(* CoDeSys 2.3 project: forGomon.pro *)
(* Libraries: esx_ioxp.lib*19.12.13 12:14:40, Standard.lib 4.10.05 11:14:46 *)

(* PLC configuration (modules and I/O channels)
gq_Ignition AT %IX0.0 [X_SYS_IGNITION] Ignition pin (D+)
gs16_TempBoard AT %IW1 [X_SYS_TEMP_BOARD] System temperature in degree Celsius
gu32_TimeMs AT %ID1 [X_SYS_TIME_MS] System time in ms
gq_StayAlive AT %QX0.0 [X_SYS_STAY_ALIVE] Stay alive mechanism
gq_Relay AT %QX1.0 [X_SYS_RELAY_1] Safety relay
gs32_SensorSupply AT %QD1 [X_SYS_SENSOR_SUPPLY_1] External sensor supply
gs32_IO01 AT %QD2 [InOut] IO01, PIN 9 (PWM H/L, DO, CC, VIN (40V), DIN) {InOut_Type = uninitialized; InOut_FilterConfig = 0; InOut_Circuit1 = X_IN_CIRCUIT_ACTIVE_HIGH; InOut_Circuit2 = X_IN_CIRCUIT_NO_PULL_UP; PWM_MaxValue = 10000}
gs32_IO02 AT %QD3 [InOut] IO02, PIN 8 (PWM H/L, DO, CC, VIN (40V), DIN) {InOut_Type = uninitialized; InOut_FilterConfig = 0; InOut_Circuit1 = X_IN_CIRCUIT_ACTIVE_HIGH; InOut_Circuit2 = X_IN_CIRCUIT_NO_PULL_UP; PWM_MaxValue = 10000}
gs32_IO03 AT %QD4 [InOut] IO03, PIN 7 (PWM H/L, DO, CC, VIN (40V), DIN) {InOut_Type = uninitialized; InOut_FilterConfig = 0; InOut_Circuit1 = X_IN_CIRCUIT_ACTIVE_HIGH; InOut_Circuit2 = X_IN_CIRCUIT_NO_PULL_UP; PWM_MaxValue = 10000}
gs32_IO04 AT %QD5 [InOut] IO04, PIN 6 (PWM H/L, DO, CC, VIN (40V), DIN) {InOut_Type = uninitialized; InOut_FilterConfig = 0; InOut_Circuit1 = X_IN_CIRCUIT_ACTIVE_HIGH; InOut_Circuit2 = X_IN_CIRCUIT_NO_PULL_UP; PWM_MaxValue = 10000}
gs32_IO05 AT %QD6 [InOut] IO05, PIN 13 (PWM H, DO, DIN) {InOut_Type = uninitialized; InOut_FilterConfig = 0; InOut_Circuit1 = X_IN_CIRCUIT_ACTIVE_HIGH; InOut_Circuit2 = X_IN_CIRCUIT_NO_PULL_UP; PWM_MaxValue = 10000}
gs32_IO06 AT %QD7 [InOut] IO06, PIN 12 (PWM H, DO, DIN) {InOut_Type = uninitialized; InOut_FilterConfig = 0; InOut_Circuit1 = X_IN_CIRCUIT_ACTIVE_HIGH; InOut_Circuit2 = X_IN_CIRCUIT_NO_PULL_UP; PWM_MaxValue = 10000}
gs32_IO07 AT %QD8 [InOut] IO07, PIN 11 (PWM H, DO, DIN) {InOut_Type = uninitialized; InOut_FilterConfig = 0; InOut_Circuit1 = X_IN_CIRCUIT_ACTIVE_HIGH; InOut_Circuit2 = X_IN_CIRCUIT_NO_PULL_UP; PWM_MaxValue = 10000}
gs32_IO08 AT %QD9 [InOut] IO08, PIN 10 (PWM H, DO, DIN) {InOut_Type = uninitialized; InOut_FilterConfig = 0; InOut_Circuit1 = X_IN_CIRCUIT_ACTIVE_HIGH; InOut_Circuit2 = X_IN_CIRCUIT_NO_PULL_UP; PWM_MaxValue = 10000}
gs32_IO09 AT %ID2 [InOut] IO09, PIN 2 (DIN, FIN, IIN) {InOut_Type = uninitialized; InOut_FilterConfig = 0; InOut_Circuit1 = X_IN_CIRCUIT_ACTIVE_HIGH; InOut_Circuit2 = X_IN_CIRCUIT_NO_PULL_UP; PWM_MaxValue = 10000}
gs32_IO10 AT %ID3 [InOut] IO10, PIN 3 (DIN, FIN, IIN) {InOut_Type = uninitialized; InOut_FilterConfig = 0; InOut_Circuit1 = X_IN_CIRCUIT_ACTIVE_HIGH; InOut_Circuit2 = X_IN_CIRCUIT_NO_PULL_UP; PWM_MaxValue = 10000}
gs32_IO11 AT %ID4 [InOut] IO11, PIN 4 (DIN, FIN, IIN) {InOut_Type = uninitialized; InOut_FilterConfig = 0; InOut_Circuit1 = X_IN_CIRCUIT_ACTIVE_HIGH; InOut_Circuit2 = X_IN_CIRCUIT_NO_PULL_UP; PWM_MaxValue = 10000}
gs32_IO12 AT %ID5 [InOut] IO12, PIN 5 (DIN) {InOut_Type = uninitialized; InOut_FilterConfig = 0; InOut_Circuit1 = X_IN_CIRCUIT_ACTIVE_HIGH; InOut_Circuit2 = X_IN_CIRCUIT_NO_PULL_UP; PWM_MaxValue = 10000}
gs32_IO13 AT %ID6 [InOut] IO13, PIN 38 (CIN (20mA), DIN) {InOut_Type = uninitialized; InOut_FilterConfig = 0; InOut_Circuit1 = X_IN_CIRCUIT_ACTIVE_HIGH; InOut_Circuit2 = X_IN_CIRCUIT_NO_PULL_UP; PWM_MaxValue = 10000}
gs32_IO14 AT %ID7 [InOut] IO14, PIN 24 (CIN (20mA), DIN) {InOut_Type = uninitialized; InOut_FilterConfig = 0; InOut_Circuit1 = X_IN_CIRCUIT_ACTIVE_HIGH; InOut_Circuit2 = X_IN_CIRCUIT_NO_PULL_UP; PWM_MaxValue = 10000}
gs32_IO15 AT %ID8 [InOut] IO15, PIN 39 (CIN (20mA), DIN) {InOut_Type = uninitialized; InOut_FilterConfig = 0; InOut_Circuit1 = X_IN_CIRCUIT_ACTIVE_HIGH; InOut_Circuit2 = X_IN_CIRCUIT_NO_PULL_UP; PWM_MaxValue = 10000}
gs32_IO16 AT %ID9 [InOut] IO16, PIN 25 (CIN (20mA), DIN) {InOut_Type = uninitialized; InOut_FilterConfig = 0; InOut_Circuit1 = X_IN_CIRCUIT_ACTIVE_HIGH; InOut_Circuit2 = X_IN_CIRCUIT_NO_PULL_UP; PWM_MaxValue = 10000}
gs32_IO17 AT %ID10 [InOut] IO17, PIN 40 (CIN (20mA), DIN) {InOut_Type = uninitialized; InOut_FilterConfig = 0; InOut_Circuit1 = X_IN_CIRCUIT_ACTIVE_HIGH; InOut_Circuit2 = X_IN_CIRCUIT_NO_PULL_UP; PWM_MaxValue = 10000}
gs32_IO18 AT %ID11 [InOut] IO18, PIN 26 (CIN (20mA), DIN) {InOut_Type = uninitialized; InOut_FilterConfig = 0; InOut_Circuit1 = X_IN_CIRCUIT_ACTIVE_HIGH; InOut_Circuit2 = X_IN_CIRCUIT_NO_PULL_UP; PWM_MaxValue = 10000}
gs32_IO19 AT %ID12 [InOut] IO19, PIN 41 (CIN (20mA), DIN) {InOut_Type = uninitialized; InOut_FilterConfig = 0; InOut_Circuit1 = X_IN_CIRCUIT_ACTIVE_HIGH; InOut_Circuit2 = X_IN_CIRCUIT_NO_PULL_UP; PWM_MaxValue = 10000}
gs32_IO20 AT %ID13 [InOut] IO20, PIN 27 (CIN (20mA), DIN) {InOut_Type = uninitialized; InOut_FilterConfig = 0; InOut_Circuit1 = X_IN_CIRCUIT_ACTIVE_HIGH; InOut_Circuit2 = X_IN_CIRCUIT_NO_PULL_UP; PWM_MaxValue = 10000}
gs32_IO21 AT %ID14 [InOut] IO21, PIN 34 (VIN (10V), DIN) {InOut_Type = uninitialized; InOut_FilterConfig = 0; InOut_Circuit1 = X_IN_CIRCUIT_ACTIVE_HIGH; InOut_Circuit2 = X_IN_CIRCUIT_NO_PULL_UP; PWM_MaxValue = 10000}
gs32_IO22 AT %ID15 [InOut] IO22, PIN 20 (VIN (10V), DIN) {InOut_Type = uninitialized; InOut_FilterConfig = 0; InOut_Circuit1 = X_IN_CIRCUIT_ACTIVE_HIGH; InOut_Circuit2 = X_IN_CIRCUIT_NO_PULL_UP; PWM_MaxValue = 10000}
gs32_IO23 AT %ID16 [InOut] IO23, PIN 35 (VIN (10V), DIN) {InOut_Type = uninitialized; InOut_FilterConfig = 0; InOut_Circuit1 = X_IN_CIRCUIT_ACTIVE_HIGH; InOut_Circuit2 = X_IN_CIRCUIT_NO_PULL_UP; PWM_MaxValue = 10000}
gs32_IO24 AT %ID17 [InOut] IO24, PIN 21 (VIN (10V), DIN) {InOut_Type = uninitialized; InOut_FilterConfig = 0; InOut_Circuit1 = X_IN_CIRCUIT_ACTIVE_HIGH; InOut_Circuit2 = X_IN_CIRCUIT_NO_PULL_UP; PWM_MaxValue = 10000}
gs32_IO25 AT %ID18 [InOut] IO25, PIN 36 (VIN (10V), DIN) {InOut_Type = uninitialized; InOut_FilterConfig = 0; InOut_Circuit1 = X_IN_CIRCUIT_ACTIVE_HIGH; InOut_Circuit2 = X_IN_CIRCUIT_NO_PULL_UP; PWM_MaxValue = 10000}
gs32_IO26 AT %ID19 [InOut] IO26, PIN 22 (VIN (10V), DIN) {InOut_Type = uninitialized; InOut_FilterConfig = 0; InOut_Circuit1 = X_IN_CIRCUIT_ACTIVE_HIGH; InOut_Circuit2 = X_IN_CIRCUIT_NO_PULL_UP; PWM_MaxValue = 10000}
RS232 [X_SER_1] node 1, in %IB80 out %QB40 {X_SER_BITRATE = 19200; X_SER_STOPBITS = 1; X_SER_MODE = 8 data bits - no parity; X_SER_RX_BUFSIZE = 256; X_SER_TX_BUFSIZE = 256}
CAN1 [X_CAN_BUS_1_XC2] node 2, in %IB80 out %QB40 {X_CAN_BUS_BITRATE = 250000; X_CAN_BUS_11BIT_MASK = 16#7FF; X_CAN_BUS_29BIT_MASK = 16#1FFFFFFF}
CAN2 [X_CAN_BUS_2_XC2] node 3, in %IB80 out %QB40 {X_CAN_BUS_BITRATE = 250000; X_CAN_BUS_11BIT_MASK = 16#7FF; X_CAN_BUS_29BIT_MASK = 16#1FFFFFFF}
*)

(* POU PLC_PRG, ST *)
PROGRAM PLC_PRG
VAR
	q_FirstCycle	: BOOL := TRUE;
	fb_SysClose		: FB_x_sys_close;
	fb_SsvTrigger	: FB_x_ssv_trigger;
END_VAR
IF (q_FirstCycle = TRUE) THEN
	q_FirstCycle := FALSE;

	(* activate 'Safety relay' *)
	gq_Relay := TRUE;

	(* activate 'Stay alive' mechanism *)
	gq_StayAlive := TRUE;

	(* activate 'Sensor Supply' *)
	gs32_SensorSupply := X_SYS_SENSOR_SUPPLY_10V;
END_IF

(* trigger 'System Supervisor' *)
fb_SsvTrigger(ou16_TriggerType:=X_SSV_TRIGGER);


IF (gq_Ignition = FALSE) THEN
	(* Ignition (D+) was switched off *)

	(* close ESX-IOXp properly *)
	fb_SysClose();
END_IF
END_PROGRAM
